DATA_BLOCK "DB_DM_PLC_VERSION"
TITLE =
//$Revision: 1.6 $
//$Date: 2007/09/06 07:44:43CEST $
//$Author: hgc $
AUTHOR : ha
FAMILY : DMG
NAME : _VERSION
VERSION : 1.1


  STRUCT
   _USERVERSION : STRING  [64 ];
  END_STRUCT ;
BEGIN
   _USERVERSION := '3S0000_SCHR_03n3';
END_DATA_BLOCK

